PROGRAM PRG_Task2
VAR
END_VAR

F_ConsumeTime(2000);

END_PROGRAM

(* stored: Version 1.1.0.1, ProductVersion 3.1.4026.18
   POU PRG_Task2: Id {d9492a9b-876f-4020-9895-a530e1a53cfe}, SpecialFunc None *)
